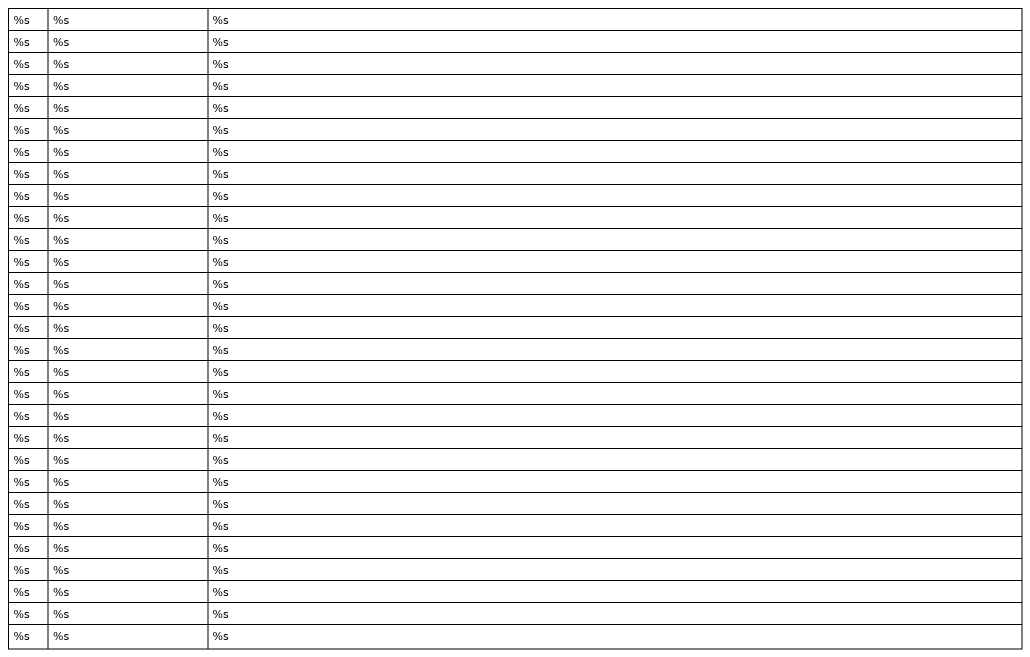
[picture p214: ZLIB_ERRORLIST (HMI screen)]
embedded screen at (0,0)-(1014,25): zLib_ErrorLine
embedded screen at (0,22)-(1014,47): zLib_ErrorLine
embedded screen at (0,44)-(1014,69): zLib_ErrorLine
embedded screen at (0,66)-(1014,91): zLib_ErrorLine
embedded screen at (0,88)-(1014,113): zLib_ErrorLine
embedded screen at (0,110)-(1014,135): zLib_ErrorLine
embedded screen at (0,132)-(1014,157): zLib_ErrorLine
embedded screen at (0,154)-(1014,179): zLib_ErrorLine
embedded screen at (0,176)-(1014,201): zLib_ErrorLine
embedded screen at (0,198)-(1014,223): zLib_ErrorLine
embedded screen at (0,220)-(1014,245): zLib_ErrorLine
embedded screen at (0,242)-(1014,267): zLib_ErrorLine
embedded screen at (0,264)-(1014,289): zLib_ErrorLine
embedded screen at (0,286)-(1014,311): zLib_ErrorLine
embedded screen at (0,308)-(1014,333): zLib_ErrorLine
embedded screen at (0,330)-(1014,355): zLib_ErrorLine
embedded screen at (0,352)-(1014,377): zLib_ErrorLine
embedded screen at (0,374)-(1014,399): zLib_ErrorLine
embedded screen at (0,396)-(1014,421): zLib_ErrorLine
embedded screen at (0,418)-(1014,443): zLib_ErrorLine
embedded screen at (0,440)-(1014,465): zLib_ErrorLine
embedded screen at (0,462)-(1014,487): zLib_ErrorLine
embedded screen at (0,484)-(1014,509): zLib_ErrorLine
embedded screen at (0,506)-(1014,531): zLib_ErrorLine
embedded screen at (0,528)-(1014,553): zLib_ErrorLine
embedded screen at (0,550)-(1014,575): zLib_ErrorLine
embedded screen at (0,572)-(1014,597): zLib_ErrorLine
embedded screen at (0,594)-(1014,619): zLib_ErrorLine
embedded screen at (0,616)-(1014,641): zLib_ErrorLine
*)

(* Visualisation VANAIN
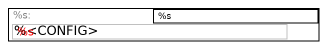
rectangle at (0,0)-(311,33): text "%s:"; shows $Object$.BitInName
rectangle at (0,12)-(281,33): text "%<CONFIG>"; shows $Object$.InstName
rectangle at (4,16)-(279,31): text "%s"; shows $Object$.ErrorString; invisible if NOT $Object$.ErrorPresent
rectangle at (145,1)-(310,15): text "%s"; shows $Object$.AnaInValue; dynamic style TRUE
*)

(* Visualisation VENCODER
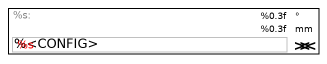
rectangle at (0,0)-(311,46): text "%s:"; shows $Object$.BitInName; alarm colour if $Object$.ErrorPresent
rectangle at (0,25)-(281,46): text "%<CONFIG>"; shows $Object$.InstName
rectangle at (4,29)-(279,44): text "%s"; shows $Object$.ErrorString; invisible if NOT $Object$.ErrorPresent OR TRUE
rectangle at (142,1)-(283,15): text "%0.3f"; shows $Object$.rpmValue * 360; dynamic style TRUE
rectangle at (282,1)-(311,15): text "°"
rectangle at (142,14)-(283,28): text "%0.3f"; shows $Object$.PosValue; dynamic style TRUE
rectangle at (282,14)-(311,28): text "mm"; invisible if $Object$.sInit.lr_LaengeProRpm = 0
rectangle at (282,25)-(312,50): text ">"; invisible if $Object$.Drehrichtung <> 1
rectangle at (282,25)-(312,50): text "<"; invisible if $Object$.Drehrichtung <> -1
rectangle at (282,25)-(312,50): text "><"; invisible if $Object$.Drehrichtung <> 0; alarm colour if $Object$.Reset; taps $Object$.Reset
*)

(* Visualisation ZLIB_ANA_IN
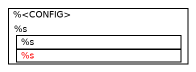
rectangle at (0,0)-(180,56): text "%<CONFIG>"; shows $Object$.InstName
rectangle at (1,14)-(166,28): text "%s"; shows $Object$.BitInName; dynamic style TRUE
rectangle at (8,41)-(173,54): text "%s"; shows $Object$.ErrorString; invisible if $Object$.ErrorString=''
rectangle at (8,27)-(173,41): text "%s"; shows $Object$.AnaInValue; dynamic style TRUE
*)

(* Visualisation ZLIB_ENCODER_IN
rectangle at (0,0)-(180,69): text "%<CONFIG>"; shows $Object$.InstName
rectangle at (1,14)-(151,28): text "%s"; shows $Object$.BitInName; dynamic style TRUE
rectangle at (8,54)-(173,67): text "%s"; shows $Object$.ErrorString; invisible if $Object$.ErrorString=''
rectangle at (10,27)-(151,41): text "%0.3f"; shows $Object$.rpmValue; dynamic style TRUE
rectangle at (150,27)-(179,41): text "°"
rectangle at (10,40)-(151,54): text "%0.3f"; shows $Object$.PosValue; dynamic style TRUE
rectangle at (150,40)-(179,54): text "mm"; invisible if $Object$.sInit.lr_LaengeProRpm = 0
rectangle at (0,0)-(30,25): text ">"; invisible if $Object$.Drehrichtung <> 1
rectangle at (0,0)-(30,25): text "<"; invisible if $Object$.Drehrichtung <> -1
rectangle at (0,0)-(30,25): text "><"; invisible if $Object$.Drehrichtung <> 0
*)

(* Visualisation VDIGIN
rectangle at (0,0)-(311,33): text "%s:"; shows $Object$.BitInName
rectangle at (0,12)-(281,33): text "%<CONFIG>"; shows $Object$.InstName
rectangle at (0,16)-(283,31): text "%s"; shows $Object$.ErrorString; invisible if NOT $Object$.ErrorPresent OR TRUE; alarm colour if $Object$.ErrorPresent
ellipse at (0,0)-(27,27): alarm colour if $Object$.BitInToCheck; tooltip $Object$
ellipse at (14,5)-(21,12): invisible if NOT $Object$.BitInToCheck
*)

(* Visualisation ZLIB_DIG_IN
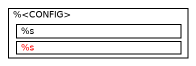
rectangle at (0,0)-(180,50): text "%<CONFIG>"; shows $Object$.InstName
rectangle at (8,16)-(173,30): text "%s"; shows $Object$.BitInName; alarm colour if $Object$.BitInToCheck; dynamic style TRUE
rectangle at (8,33)-(173,46): text "%s"; shows $Object$.ErrorString; invisible if NOT $Object$.ErrorPresent
*)

(* Visualisation ZLIB_SENSORCHECK
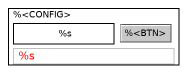
rectangle at (0,0)-(171,57): text "%<CONFIG>"; shows $Object$.InstName
rectangle at (5,15)-(106,36): text "%s"; shows $Object$.BitInName; alarm colour if $Object$.BitInToCheck; dynamic style TRUE
rectangle at (5,40)-(166,56): text "%s"; shows $Object$.ErrorString; invisible if NOT $Object$.ErrorPresent
button at (112,16)-(163,34): text "%<BTN>"; shows $Object$.BtnReset.Text; invisible if NOT $Object$.BtnReset.Visible; taps $Object$.BtnReset.Pressed; dynamic style $Object$.BtnReset.TextColor, $Object$.BtnReset.BackgroundColor, $Object$.BtnReset.BackgroundColor, NOT $Object$.BtnReset.Enable
*)

(* Visualisation VBTN_SMAL
rounded rectangle at (0,0)-(51,51): shows $Object$.Text; invisible if NOT $Object$.Visible; taps $Object$.Pressed; dynamic style $Object$.TextColor, NOT $Object$.Enable
*)

(* Visualisation VDIGOUT
rectangle at (0,0)-(361,75): text "%s:"; shows $Object$.InstName
rectangle at (2,12)-(361,33): text "%<CONFIG>"; shows $Object$.InstName
embedded screen at (142,30)-(271,73): ZLIB_VISUBUTTON
ellipse at (0,0)-(27,27): alarm colour if $Object$.BitOutToSet
ellipse at (15,4)-(22,11): invisible if NOT $Object$.BitOutToSet
embedded screen at (11,30)-(140,73): ZLIB_VISUBUTTON
*)

(* Visualisation VDIGOUT_SMAL
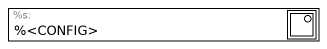
rectangle at (0,0)-(311,33): text "%s:"; shows $Object$.InstName; tooltip $Object$
rectangle at (0,12)-(311,33): text "%<CONFIG>"; shows $Object$.InstName; tooltip $Object$
rounded rectangle at (279,2)-(308,31): alarm colour if NOT $Object$.BtnOutput.Enable
rounded rectangle at (282,5)-(305,28): alarm colour if $Object$.BitOutToSet
ellipse at (296,7)-(303,14): invisible if NOT $Object$.BitOutToSet
embedded screen at (0,2)-(311,31): VBtn_smal; invisible if $Object$.BitOutToSet; tooltip $Object$; dynamic style $Object$.Disabled
embedded screen at (0,2)-(311,31): VBtn_smal; invisible if NOT $Object$.BitOutToSet; tooltip $Object$; dynamic style $Object$.Disabled
*)

(* Visualisation ZLIB_DIGOUT
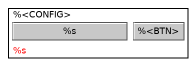
rectangle at (0,0)-(180,50): text "%<CONFIG>"; shows $Object$.InstName; alarm colour if $Object$.BitOutToSet
rounded rectangle at (0,36)-(177,50): text "%s"; shows $Object$.ErrorString; invisible if NOT $Object$.ErrorPresent
button at (125,14)-(176,32): text "%<BTN>"; shows $Object$.BtnReset.Text; invisible if NOT $Object$.BtnReset.Visible; taps $Object$.BtnReset.Pressed; dynamic style $Object$.BtnReset.TextColor, $Object$.BtnReset.BackgroundColor, $Object$.BtnReset.BackgroundColor, NOT $Object$.BtnReset.Enable
button at (4,14)-(119,32): text "%s"; shows $Object$.BtnOutput.Text; invisible if NOT $Object$.BtnOutput.Visible; taps $Object$.BtnOutput.Pressed; dynamic style $Object$.BtnOutput.TextColor, $Object$.BtnOutput.BackgroundColor, $Object$.BtnOutput.BackgroundColor, NOT $Object$.BtnOutput.Enable
*)

(* Visualisation ZLIB_DIGOUTIN
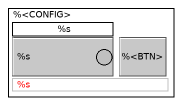
rectangle at (0,0)-(166,89): text "%<CONFIG>"; shows $Object$.InstName
rectangle at (4,14)-(105,28): text "%s"; shows $Object$.BitInName; invisible if NOT($Object$.InputAvailable); alarm colour if $Object$.BitInToCheck; dynamic style TRUE
rounded rectangle at (4,70)-(160,83): text "%s"; shows $Object$.ErrorString; invisible if NOT $Object$.ErrorPresent
button at (111,29)-(158,68): text "%<BTN>"; shows $Object$.BtnReset.Text; invisible if NOT $Object$.BtnReset.Visible; taps $Object$.BtnReset.Pressed; dynamic style $Object$.BtnReset.TextColor, $Object$.BtnReset.BackgroundColor, $Object$.BtnReset.BackgroundColor, NOT $Object$.BtnReset.Enable
button at (4,29)-(105,68): text "%s"; shows $Object$.BtnOutput.Text; invisible if NOT $Object$.BtnOutput.Visible; taps $Object$.BtnOutput.Pressed; dynamic style $Object$.BtnOutput.TextColor, $Object$.BtnOutput.BackgroundColor, $Object$.BtnOutput.BackgroundColor, NOT $Object$.BtnOutput.Enable
ellipse at (88,41)-(104,57): invisible if NOT($Object$.BtnOutput.Visible); alarm colour if $Object$.BitOutToSet
*)

(* Visualisation ZLIB_EPSON_DETAILS
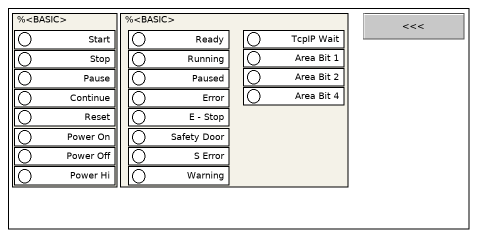
rectangle at (4,5)-(109,179): text "%<BASIC>"; shows 'RoboInput'
rectangle at (112,5)-(340,179): text "%<BASIC>"; shows 'RoboOutput'
rectangle at (6,22)-(107,41): text "Start"
ellipse at (10,24)-(23,38): alarm colour if $Object$.RemOutStart
rectangle at (6,42)-(107,60): text "Stop"
ellipse at (10,44)-(23,58): alarm colour if $Object$.RemOutStop
rectangle at (6,61)-(107,80): text "Pause"
ellipse at (10,63)-(23,77): alarm colour if $Object$.RemOutPause
rectangle at (6,81)-(107,99): text "Continue"
ellipse at (10,83)-(23,97): alarm colour if $Object$.RemOutCont
rectangle at (6,100)-(107,118): text "Reset"
ellipse at (10,102)-(23,116): alarm colour if $Object$.RemOutReset
rectangle at (6,120)-(107,138): text "Power On"
ellipse at (10,122)-(23,136): alarm colour if $Object$.RemOutPowerOn
rectangle at (6,139)-(107,157): text "Power Off"
ellipse at (10,141)-(23,155): alarm colour if $Object$.RemOutPowerOff
rectangle at (6,158)-(107,177): text "Power Hi"
ellipse at (10,161)-(23,175): alarm colour if $Object$.RemOutPowerHi
rectangle at (120,22)-(221,41): text "Ready"
ellipse at (124,24)-(137,38): alarm colour if $Object$.RemInReady
rectangle at (120,42)-(221,60): text "Running"
ellipse at (124,44)-(137,58): alarm colour if $Object$.RemInRunning
rectangle at (120,61)-(221,80): text "Paused"
ellipse at (124,63)-(137,77): alarm colour if $Object$.RemInPaused
rectangle at (120,81)-(221,99): text "Error"
ellipse at (124,83)-(137,97): alarm colour if $Object$.RemInError
rectangle at (120,100)-(221,118): text "E - Stop"
ellipse at (124,102)-(137,116): alarm colour if $Object$.RemInEStopOn
rectangle at (120,120)-(221,138): text "Safety Door"
ellipse at (124,122)-(137,136): alarm colour if $Object$.RemInSafeguardOn
rectangle at (120,139)-(221,157): text "S Error"
ellipse at (124,141)-(137,155): alarm colour if $Object$.RemInSError
rectangle at (120,158)-(221,177): text "Warning"
ellipse at (124,161)-(137,175): alarm colour if $Object$.RemInWarning
rectangle at (235,41)-(336,59): text "Area Bit 1"
ellipse at (239,43)-(252,57): alarm colour if $Object$.RemInAreaBit1
rectangle at (235,60)-(336,78): text "Area Bit 2"
ellipse at (239,62)-(252,76): alarm colour if $Object$.RemInAreaBit2
rectangle at (235,79)-(336,97): text "Area Bit 4"
ellipse at (239,81)-(252,95): alarm colour if $Object$.RemInAreaBit4
rectangle at (235,22)-(336,40): text "TcpIP Wait"
ellipse at (239,24)-(252,38): alarm colour if $Object$.RemInTcpIP_Wait
button at (355,5)-(456,31): text "<<<"; toggles $Object$.ShowDetails; dynamic style color.lightgrey
1 more shapes without text or variables
*)

(* Visualisation ZLIB_EPSON_POSLIST
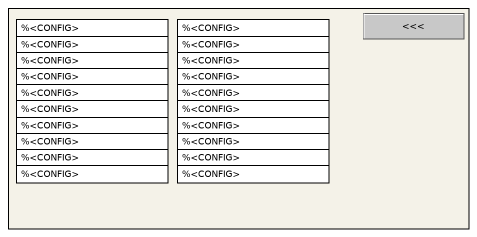
button at (355,5)-(456,31): text "<<<"; toggles $Object$.ShowPosArray; dynamic style color.lightgrey
rectangle at (169,11)-(321,29): text "%<CONFIG>"; shows $Object$.PosArray[11]
rectangle at (169,28)-(321,45): text "%<CONFIG>"; shows $Object$.PosArray[12]
rectangle at (169,44)-(321,61): text "%<CONFIG>"; shows $Object$.PosArray[13]
rectangle at (169,60)-(321,77): text "%<CONFIG>"; shows $Object$.PosArray[14]
rectangle at (169,76)-(321,94): text "%<CONFIG>"; shows $Object$.PosArray[15]
rectangle at (169,92)-(321,110): text "%<CONFIG>"; shows $Object$.PosArray[16]
rectangle at (169,109)-(321,126): text "%<CONFIG>"; shows $Object$.PosArray[17]
rectangle at (169,125)-(321,142): text "%<CONFIG>"; shows $Object$.PosArray[18]
rectangle at (169,141)-(321,158): text "%<CONFIG>"; shows $Object$.PosArray[19]
rectangle at (169,157)-(321,175): text "%<CONFIG>"; shows $Object$.PosArray[20]
rectangle at (8,11)-(160,29): text "%<CONFIG>"; shows $Object$.PosArray[1]
rectangle at (8,28)-(160,45): text "%<CONFIG>"; shows $Object$.PosArray[2]
rectangle at (8,44)-(160,61): text "%<CONFIG>"; shows $Object$.PosArray[3]
rectangle at (8,60)-(160,77): text "%<CONFIG>"; shows $Object$.PosArray[4]
rectangle at (8,76)-(160,94): text "%<CONFIG>"; shows $Object$.PosArray[5]
rectangle at (8,92)-(160,110): text "%<CONFIG>"; shows $Object$.PosArray[6]
rectangle at (8,109)-(160,126): text "%<CONFIG>"; shows $Object$.PosArray[7]
rectangle at (8,125)-(160,142): text "%<CONFIG>"; shows $Object$.PosArray[8]
rectangle at (8,141)-(160,158): text "%<CONFIG>"; shows $Object$.PosArray[9]
rectangle at (8,157)-(160,175): text "%<CONFIG>"; shows $Object$.PosArray[10]
1 more shapes without text or variables
*)

(* Visualisation ZLIB_EPSON_ROBOT
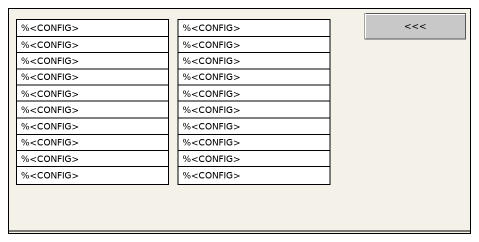
embedded screen at (0,0)-(463,226): ZLIB_EPSON_Steuerung
embedded screen at (0,0)-(463,223): ZLIB_EPSON_DETAILS; invisible if NOT $Object$.ShowDetails
embedded screen at (0,0)-(463,223): ZLIB_EPSON_POSLIST; invisible if NOT $Object$.ShowPosArray
*)

(* Visualisation ZLIB_EPSON_STEUERUNG
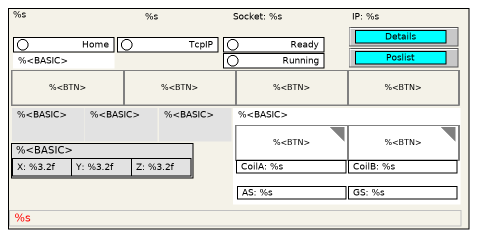
rectangle at (0,0)-(461,221): text "%s"; shows $Object$.BitName
rectangle at (215,29)-(316,44): text "Ready"
ellipse at (219,31)-(230,42): alarm colour if $Object$.RemInReady
rectangle at (215,45)-(316,60): text "Running"
ellipse at (219,47)-(230,58): alarm colour if $Object$.RemInRunning
rectangle at (5,45)-(106,60): text "%d"; shows $Object$.ActualArea
embedded screen at (3,62)-(116,97): ZLIB_VISUBUTTON
rectangle at (1,202)-(453,218): text "%s"; shows $Object$.ErrorString; invisible if $Object$.ErrorPresent
rectangle at (69,2)-(218,15): text "%s"; shows $Object$.Description
embedded screen at (339,62)-(451,97): zLib_VisuButton
rectangle at (4,100)-(76,133): text "%d"; shows $Object$.PosNo; editable
rectangle at (77,100)-(149,133): text "%d"; shows $Object$.ActualPosition
embedded screen at (115,62)-(228,97): zLib_VisuButton
embedded screen at (227,62)-(340,97): zLib_VisuButton
rectangle at (5,29)-(106,44): text "Home"
ellipse at (9,31)-(20,42): alarm colour if $Object$.HomePosition
rectangle at (109,29)-(210,44): text "TcpIP"
ellipse at (113,31)-(124,42): alarm colour if $Object$.ConnectionAlive
button at (341,19)-(450,38): text "%<BTN>"; shows 'Details'; toggles $Object$.ShowDetails; dynamic style color.lightgrey
button at (341,40)-(450,59): text "%<BTN>"; shows 'Poslist'; toggles $Object$.ShowPosArray; dynamic style color.lightgrey
rectangle at (151,100)-(223,133): text "%d"; shows $Object$.PosOffset
rectangle at (225,100)-(452,196): text "%<BASIC>"; shows 'Tool'
embedded screen at (227,117)-(340,152): zLib_VisuButton
embedded screen at (339,117)-(451,152): zLib_VisuButton
rectangle at (228,152)-(338,165): text "CoilA: %s"; shows $Object$.NameCoilA; alarm colour if $Object$.RemInToolCoilA
rectangle at (340,152)-(449,165): text "CoilB: %s"; shows $Object$.NameCoilB; invisible if $Object$.NameCoilB='xxxx'; alarm colour if $Object$.RemInToolCoilB
rectangle at (340,178)-(449,191): text "GS: %s"; shows $Object$.NameInitSensor; invisible if $Object$.NameInitSensor='xxxx'; alarm colour if $Object$.RemInToolInitSensor
rectangle at (229,178)-(338,191): text "AS: %s"; shows $Object$.NameWorkSensor; invisible if $Object$.NameWorkSensor='xxxx'; alarm colour if $Object$.RemInToolWorkSensor
rectangle at (339,2)-(452,15): text "IP: %s"; shows $Object$.TcpIpAdress
rectangle at (220,2)-(338,15): text "Socket: %s"; shows $Object$.SocketState
rectangle at (347,43)-(438,56): text "Poslist"; invisible if TRUE
rectangle at (347,22)-(438,35): text "Details"; invisible if TRUE
rectangle at (3,135)-(185,170): text "%<BASIC>"; shows 'aktAchsPos'
rectangle at (4,150)-(64,168): text "X: %3.2f"; shows $Object$.PosX
rectangle at (63,150)-(124,168): text "Y: %3.2f"; shows $Object$.PosY
rectangle at (123,150)-(183,168): text "Z: %3.2f"; shows $Object$.PosZ
rectangle at (4,100)-(76,133): text "%<BASIC>"; shows 'sollPos'
rectangle at (77,100)-(149,133): text "%<BASIC>"; shows 'aktPos'
rectangle at (151,100)-(223,133): text "%<BASIC>"; shows 'aktOffset'
rectangle at (5,45)-(106,60): text "%<BASIC>"; shows 'ActualArea'
polygon at (322,119)-(336,133): alarm colour if $Object$.RemOutSetToolOn
polygon at (433,119)-(447,133): alarm colour if $Object$.RemOutSetToolOff
*)

(* Visualisation ZLIB_LOGIN
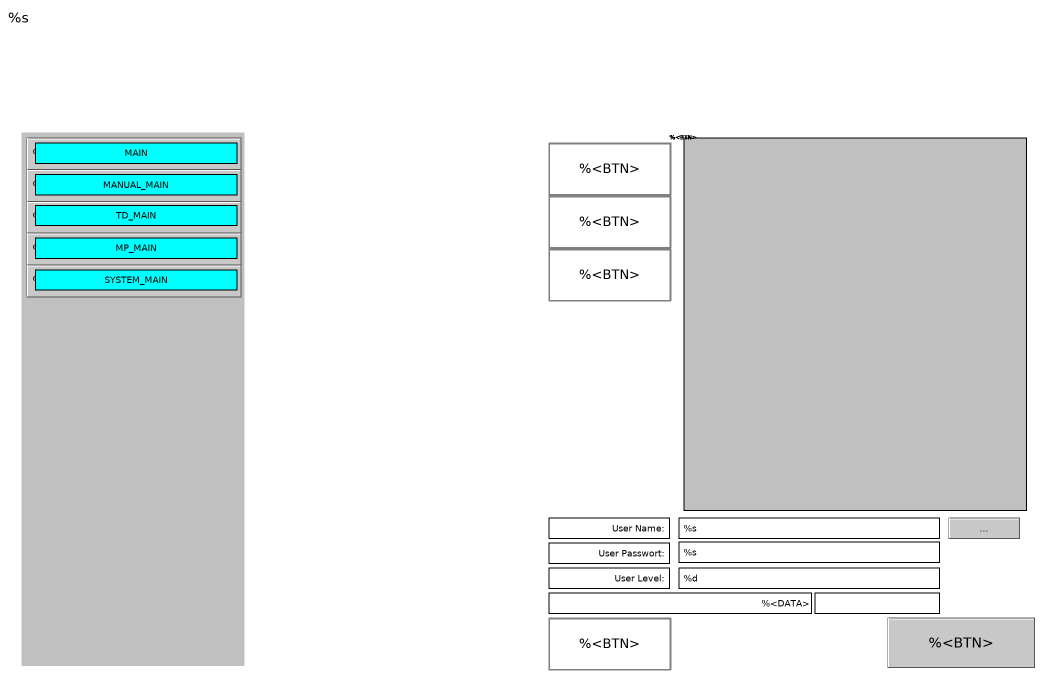
embedded screen at (530,231)-(652,283): ZLIB_VISUBUTTON
button at (869,600)-(1016,650): text "%<BTN>"; shows 'zurück'; opens ZOOMTOCALLER; dynamic style Color.lightgrey
rectangle at (0,0)-(0,0): text "%s"; shows UD.UserList[INDEX].UserName; alarm colour if $ROWCONST$ = .Visu.LoginHandler.UserListIndex
embedded screen at (530,125)-(652,177): ZLIB_VISUBUTTON
embedded screen at (530,178)-(652,230): ZLIB_VISUBUTTON
embedded screen at (665,120)-(1008,493): ZLIB_NUMERIC_KEYPAD; invisible if NOT .Visu.LoginHandler.LoginKeyPad.Visible; dynamic style NOT .Visu.LoginHandler.LoginKeyPad.Enable
rectangle at (530,500)-(651,521): text "User Name:"; invisible if NOT .Visu.LoginHandler.ShowEditFields
rectangle at (530,575)-(793,596): text "%<DATA>"; shows 'Passwort ändern'; invisible if NOT .Visu.LoginHandler.ShowEditFields
rectangle at (530,525)-(651,546): text "User Passwort:"; invisible if NOT .Visu.LoginHandler.ShowEditFields
rectangle at (530,550)-(651,571): text "User Level:"; invisible if NOT .Visu.LoginHandler.ShowEditFields
rectangle at (660,500)-(921,521): text "%s"; shows .Visu.LoginHandler.UserEdit.UserName; invisible if NOT .Visu.LoginHandler.ShowEditFields; editable
rectangle at (660,524)-(921,545): text "%s"; shows .Visu.LoginHandler.UserEdit.UserPassword; invisible if NOT .Visu.LoginHandler.ShowEditFields; editable
rectangle at (796,575)-(921,596): invisible if NOT .Visu.LoginHandler.ShowEditFields; alarm colour if .Visu.LoginHandler.UserEdit.UserCanChangeOwnPassword; toggles .Visu.LoginHandler.UserEdit.UserCanChangeOwnPassword
rectangle at (660,550)-(921,571): text "%d"; shows .Visu.LoginHandler.UserEdit.UserLevel; invisible if NOT .Visu.LoginHandler.ShowEditFields; editable 0..6
embedded screen at (530,600)-(652,652): ZLIB_VISUBUTTON
button at (930,500)-(1001,521): text "..."; shows .Visu.LoginHandler.UserEdit.UserName; invisible if NOT .Visu.LoginHandler.ShowEditFields; editable
embedded screen at (3,115)-(226,648): M0000_Main
1 more shapes without text or variables
*)

(* Visualisation ZLIB_NUMERIC_KEYPAD
rectangle at (5,4)-(314,25): text "%s"; shows $sNumericKeypad$.InputString
embedded screen at (4,26)-(79,99): ZLIB_VISUBUTTON
embedded screen at (78,26)-(153,99): ZLIB_VISUBUTTON
embedded screen at (152,26)-(227,99): ZLIB_VISUBUTTON
embedded screen at (4,98)-(79,171): ZLIB_VISUBUTTON
embedded screen at (78,98)-(153,171): ZLIB_VISUBUTTON
embedded screen at (152,98)-(227,171): ZLIB_VISUBUTTON
embedded screen at (4,170)-(79,243): ZLIB_VISUBUTTON
embedded screen at (78,170)-(153,243): ZLIB_VISUBUTTON
embedded screen at (152,242)-(227,315): ZLIB_VISUBUTTON
embedded screen at (4,242)-(79,315): ZLIB_VISUBUTTON
embedded screen at (78,242)-(153,315): ZLIB_VISUBUTTON
embedded screen at (152,170)-(227,243): ZLIB_VISUBUTTON
embedded screen at (240,26)-(315,99): ZLIB_VISUBUTTON
embedded screen at (240,98)-(315,171): ZLIB_VISUBUTTON
embedded screen at (240,170)-(315,243): ZLIB_VISUBUTTON
embedded screen at (240,242)-(315,315): ZLIB_VISUBUTTON
1 more shapes without text or variables
*)

(* Visualisation ZLIB_MESSAGELINE
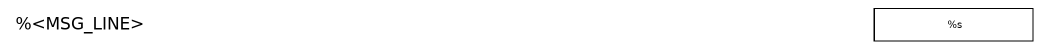
embedded screen at (0,0)-(1025,33): zLib_MessageLineBool; invisible if $MsgLine$.MsgTypeEnum <> 1
embedded screen at (0,0)-(1025,33): zLib_MessageLineDint; invisible if $MsgLine$.MsgTypeEnum <> 2
embedded screen at (0,0)-(1025,33): zLib_MessageLineReal; invisible if $MsgLine$.MsgTypeEnum <> 3
embedded screen at (0,0)-(1025,33): zLib_MessageLineString; invisible if $MsgLine$.MsgTypeEnum <> 4
*)

(* Visualisation ZLIB_MESSAGELINEBOOL
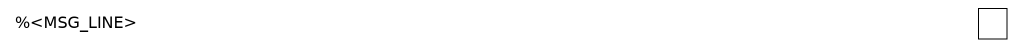
rectangle at (0,0)-(969,29): text "%<MSG_LINE>"; shows $MsgLine$.Text; invisible if NOT $MsgLine$.Visible; toggles $MsgLine$.MsgBool
rectangle at (970,0)-(999,31): invisible if NOT $MsgLine$.Visible; alarm colour if $MsgLine$.MsgBool; toggles $MsgLine$.MsgBool; dynamic style NOT $MsgLine$.Editable OR NOT $MsgLine$.Visible
*)

(* Visualisation ZLIB_MESSAGELINEDINT
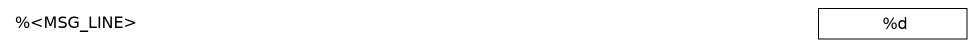
rectangle at (0,0)-(805,29): text "%<MSG_LINE>"; shows $MsgLine$.Text; invisible if NOT $MsgLine$.Visible
rectangle at (810,0)-(959,31): text "%d"; shows $MsgLine$.MsgInt; invisible if NOT $MsgLine$.Visible; editable; dynamic style NOT $MsgLine$.Editable OR NOT $MsgLine$.Visible
*)

(* Visualisation ZLIB_MESSAGELINEREAL
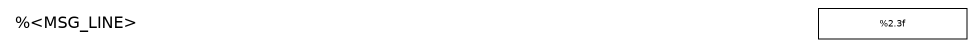
rectangle at (0,0)-(805,29): text "%<MSG_LINE>"; shows $MsgLine$.Text; invisible if NOT $MsgLine$.Visible
rectangle at (810,0)-(959,31): text "%2.3f"; shows $MsgLine$.MsgReal; invisible if NOT $MsgLine$.Visible; editable; dynamic style NOT $MsgLine$.Editable OR NOT $MsgLine$.Visible
*)

(* Visualisation ZLIB_MESSAGELINESTRING
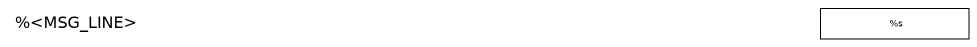
rectangle at (0,0)-(805,29): text "%<MSG_LINE>"; shows $MsgLine$.Text; invisible if NOT $MsgLine$.Visible
rectangle at (812,0)-(961,31): text "%s"; shows $MsgLine$.MsgString; invisible if NOT $MsgLine$.Visible; editable; dynamic style NOT $MsgLine$.Editable OR NOT $MsgLine$.Visible
*)

(* Visualisation ZLIB_SHOWMESSAGEBUTTON
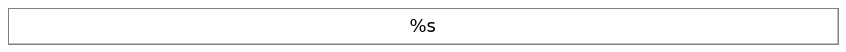
rectangle at (0,0)-(830,36): text "%s"; shows $Object$.Text; invisible if NOT $Object$.Visible; alarm colour if NOT $Object$.Enable; taps $Object$.Pressed; dynamic style $Object$.TextColor, $Object$.BackgroundColor, $Object$.BackgroundColor, NOT $Object$.Enable
polyline at (830,0)-(830,36): invisible if NOT $Object$.Visible; alarm colour if $Object$.Pressed
polyline at (0,36)-(830,36): invisible if NOT $Object$.Visible; alarm colour if $Object$.Pressed
polyline at (6,0)-(823,0): invisible if NOT $Object$.Visible; alarm colour if NOT $Object$.Pressed
polyline at (0,0)-(0,36): invisible if NOT $Object$.Visible; alarm colour if NOT $Object$.Pressed
polyline at (0,36)-(830,36): invisible if NOT $Object$.Visible; alarm colour if $Object$.Pressed
polyline at (830,0)-(830,36): invisible if NOT $Object$.Visible; alarm colour if $Object$.Pressed
polyline at (0,0)-(830,0): invisible if NOT $Object$.Visible; alarm colour if NOT $Object$.Pressed
polyline at (0,0)-(0,36): invisible if NOT $Object$.Visible; alarm colour if NOT $Object$.Pressed
*)

(* Visualisation ZLIB_VISUMESSAGEHANDLER
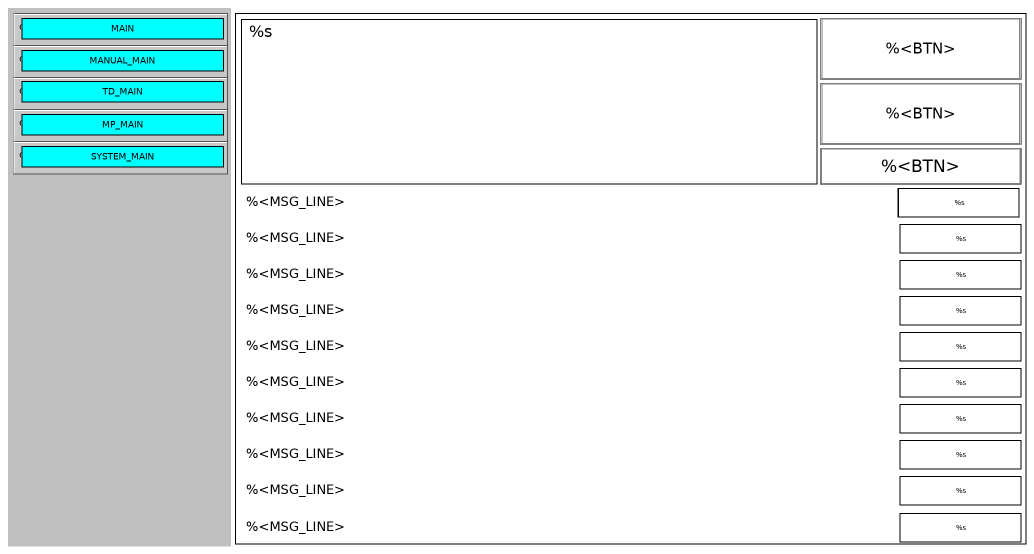
rectangle at (230,120)-(1021,651): dynamic style .Visu.Message.Color, .Visu.Message.Color
embedded screen at (815,190)-(1016,251): ZLIB_VISUBUTTON
embedded screen at (815,255)-(1016,291): ZLIB_VISUBUTTON_S17
embedded screen at (235,295)-(1014,324): zLib_MessageLine
embedded screen at (235,331)-(1016,360): zLib_MessageLine
embedded screen at (235,367)-(1016,396): zLib_MessageLine
embedded screen at (235,403)-(1016,432): zLib_MessageLine
embedded screen at (235,439)-(1016,468): zLib_MessageLine
embedded screen at (235,475)-(1016,504): zLib_MessageLine
embedded screen at (235,511)-(1016,540): zLib_MessageLine
embedded screen at (235,547)-(1016,576): zLib_MessageLine
embedded screen at (235,583)-(1016,612): zLib_MessageLine
embedded screen at (235,620)-(1016,649): zLib_MessageLine
embedded screen at (815,125)-(1016,186): ZLIB_VISUBUTTON
embedded screen at (3,115)-(226,653): M0000_Main
rectangle at (242,128)-(808,289): text "%s"; shows .Visu.Message.Text
1 more shapes without text or variables
*)

(* Visualisation ZLIB_VALVE_1_SENSORS
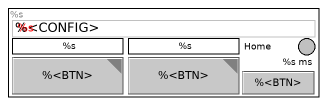
rectangle at (0,0)-(311,89): text "%s"; shows $Object$.BitName
rectangle at (4,30)-(115,46): text "%s"; shows $Object$.SAInitPosName; invisible if $Object$.NoOfInitSensors<1; alarm colour if $Object$.AInitPosition; dynamic style TRUE
rectangle at (120,30)-(231,46): text "%s"; shows $Object$.SAWorkPosName; invisible if $Object$.NoOfWorkSensors<1; alarm colour if $Object$.AWorkPosition; dynamic style TRUE
rectangle at (5,11)-(306,28): text "%<CONFIG>"; shows $Object$.InstName
button at (234,63)-(306,86): text "%<BTN>"; shows $Object$.BtnReset.Text; invisible if NOT $Object$.BtnReset.Visible; taps $Object$.BtnReset.Pressed; dynamic style $Object$.BtnReset.TextColor, $Object$.BtnReset.BackgroundColor, $Object$.BtnReset.BackgroundColor, NOT $Object$.BtnReset.Enable
button at (120,49)-(231,86): text "%<BTN>"; shows $Object$.BtnMoveWork.Text; invisible if NOT $Object$.BtnMoveWork.Visible; taps $Object$.BtnMoveWork.Pressed; dynamic style $Object$.BtnMoveWork.TextColor, $Object$.BtnMoveWork.BackgroundColor, $Object$.BtnMoveWork.BackgroundColor, NOT $Object$.BtnMoveWork.Enable
button at (4,49)-(115,86): text "%<BTN>"; shows $Object$.BtnMoveInit.Text; invisible if NOT $Object$.BtnMoveInit.Visible; taps $Object$.BtnMoveInit.Pressed; dynamic style $Object$.BtnMoveInit.TextColor, $Object$.BtnMoveInit.BackgroundColor, $Object$.BtnMoveInit.BackgroundColor, NOT $Object$.BtnMoveInit.Enable
ellipse at (290,30)-(307,47): alarm colour if $Object$.HomePosition; dynamic style TRUE
rounded rectangle at (234,32)-(280,45): text "Home"; shows $Object$.State
rectangle at (235,46)-(306,62): text "%s ms"; shows $Object$.ProcessTime
rounded rectangle at (4,12)-(307,29): text "%s"; shows $Object$.ErrorString; invisible if NOT $Object$.ErrorPresent
polygon at (99,51)-(113,65): invisible if $Object$.NoOfValveCoils<2; alarm colour if $Object$.CoilB
polygon at (215,51)-(229,65): alarm colour if $Object$.CoilA
*)

(* Visualisation ZLIB_VALVE_2_SENSORS
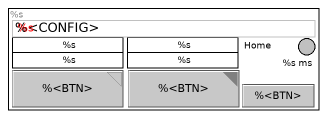
rectangle at (0,0)-(311,102): text "%s"; shows $Object$.BitName
rectangle at (4,29)-(115,45): text "%s"; shows $Object$.SAInitPosName; invisible if $Object$.NoOfInitSensors<1; alarm colour if $Object$.AInitPosition; dynamic style TRUE
rectangle at (4,44)-(115,60): text "%s"; shows $Object$.SBInitPosName; invisible if $Object$.NoOfInitSensors<2; alarm colour if $Object$.BInitPosition; dynamic style TRUE
rectangle at (119,29)-(230,45): text "%s"; shows $Object$.SAWorkPosName; invisible if $Object$.NoOfWorkSensors<1; alarm colour if $Object$.AWorkPosition; dynamic style TRUE
rectangle at (119,44)-(230,60): text "%s"; shows $Object$.SBWorkPosName; invisible if $Object$.NoOfWorkSensors<2; alarm colour if $Object$.BWorkPosition; dynamic style TRUE
button at (234,76)-(306,99): text "%<BTN>"; shows $Object$.BtnReset.Text; invisible if NOT $Object$.BtnReset.Visible; taps $Object$.BtnReset.Pressed; dynamic style $Object$.BtnReset.TextColor, $Object$.BtnReset.BackgroundColor, $Object$.BtnReset.BackgroundColor, NOT $Object$.BtnReset.Enable
button at (120,62)-(231,99): text "%<BTN>"; shows $Object$.BtnMoveWork.Text; invisible if NOT $Object$.BtnMoveWork.Visible; taps $Object$.BtnMoveWork.Pressed; dynamic style $Object$.BtnMoveWork.TextColor, $Object$.BtnMoveWork.BackgroundColor, $Object$.BtnMoveWork.BackgroundColor, NOT $Object$.BtnMoveWork.Enable
button at (4,62)-(115,99): text "%<BTN>"; shows $Object$.BtnMoveInit.Text; invisible if NOT $Object$.BtnMoveInit.Visible; taps $Object$.BtnMoveInit.Pressed; dynamic style $Object$.BtnMoveInit.TextColor, $Object$.BtnMoveInit.BackgroundColor, $Object$.BtnMoveInit.BackgroundColor, NOT $Object$.BtnMoveInit.Enable
ellipse at (290,30)-(307,47): alarm colour if $Object$.HomePosition; dynamic style TRUE
rounded rectangle at (234,31)-(280,44): text "Home"; shows $Object$.State
rectangle at (235,47)-(306,63): text "%s ms"; shows $Object$.ProcessTime
rectangle at (5,11)-(306,28): text "%<CONFIG>"; shows $Object$.InstName
rounded rectangle at (4,12)-(307,29): text "%s"; shows $Object$.ErrorString; invisible if NOT $Object$.ErrorPresent
polygon at (99,64)-(113,78): invisible if $Object$.NoOfValveCoils<2; alarm colour if $Object$.CoilB
polygon at (215,64)-(229,78): alarm colour if $Object$.CoilA
*)

(* Visualisation ZLIB_VALVE_3_SENSORS
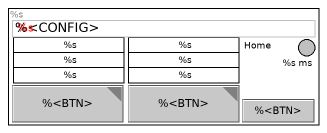
rectangle at (0,0)-(311,117): text "%s"; shows $Object$.BitName
rectangle at (5,29)-(116,45): text "%s"; shows $Object$.SAInitPosName; invisible if $Object$.NoOfInitSensors<1; alarm colour if $Object$.AInitPosition; dynamic style TRUE
rectangle at (5,44)-(116,60): text "%s"; shows $Object$.SBInitPosName; invisible if $Object$.NoOfInitSensors<2; alarm colour if $Object$.BInitPosition; dynamic style TRUE
rectangle at (120,29)-(231,45): text "%s"; shows $Object$.SAWorkPosName; invisible if $Object$.NoOfWorkSensors<1; alarm colour if $Object$.AWorkPosition; dynamic style TRUE
rectangle at (120,44)-(231,60): text "%s"; shows $Object$.SBWorkPosName; invisible if $Object$.NoOfWorkSensors<2; alarm colour if $Object$.BWorkPosition; dynamic style TRUE
ellipse at (290,31)-(307,48): alarm colour if $Object$.HomePosition; dynamic style TRUE
rounded rectangle at (234,31)-(280,44): text "Home"; shows $Object$.State
rectangle at (235,47)-(306,63): text "%s ms"; shows $Object$.ProcessTime
rectangle at (5,59)-(116,75): text "%s"; shows $Object$.SCInitPosName; invisible if $Object$.NoOfInitSensors<3; alarm colour if $Object$.CInitPosition; dynamic style TRUE
rectangle at (120,59)-(231,75): text "%s"; shows $Object$.SCWorkPosName; invisible if $Object$.NoOfWorkSensors<3; alarm colour if $Object$.CWorkPosition; dynamic style TRUE
button at (234,91)-(306,114): text "%<BTN>"; shows $Object$.BtnReset.Text; invisible if NOT $Object$.BtnReset.Visible; taps $Object$.BtnReset.Pressed; dynamic style $Object$.BtnReset.TextColor, $Object$.BtnReset.BackgroundColor, $Object$.BtnReset.BackgroundColor, NOT $Object$.BtnReset.Enable
button at (120,77)-(231,114): text "%<BTN>"; shows $Object$.BtnMoveWork.Text; invisible if NOT $Object$.BtnMoveWork.Visible; taps $Object$.BtnMoveWork.Pressed; dynamic style $Object$.BtnMoveWork.TextColor, $Object$.BtnMoveWork.BackgroundColor, $Object$.BtnMoveWork.BackgroundColor, NOT $Object$.BtnMoveWork.Enable
button at (4,77)-(115,114): text "%<BTN>"; shows $Object$.BtnMoveInit.Text; invisible if NOT $Object$.BtnMoveInit.Visible; taps $Object$.BtnMoveInit.Pressed; dynamic style $Object$.BtnMoveInit.TextColor, $Object$.BtnMoveInit.BackgroundColor, $Object$.BtnMoveInit.BackgroundColor, NOT $Object$.BtnMoveInit.Enable
rectangle at (5,11)-(306,28): text "%<CONFIG>"; shows $Object$.InstName
rounded rectangle at (4,12)-(307,29): text "%s"; shows $Object$.ErrorString; invisible if NOT $Object$.ErrorPresent
polygon at (99,79)-(113,93): invisible if $Object$.NoOfValveCoils<2; alarm colour if $Object$.CoilB
polygon at (215,79)-(229,93): alarm colour if $Object$.CoilA
*)

(* Visualisation ZLIB_VALVE_5_SENSORS
